PROGRAM VarPersistentes
VAR
		Datos_persistentes :WritePersistentData;
		StartON:TON;
		IntervalON:TON;
END_VAR
VAR // added by the converter: edge detectors and wires of the graphical bodies
    _rt1 : R_TRIG;
END_VAR

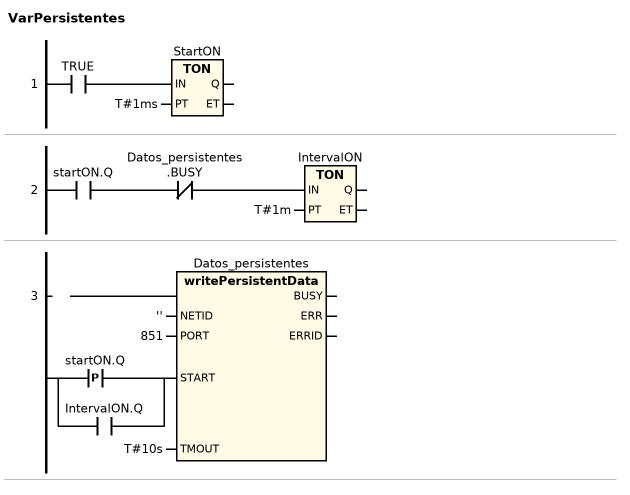
// NETWORK 1
StartON(IN := TRUE, PT := T#1ms); // TON

// NETWORK 2
IntervalON(IN := startON.Q AND NOT Datos_persistentes.BUSY, PT := T#1m); // TON

// NETWORK 3
_rt1(CLK := startON.Q);
Datos_persistentes(NETID := '', PORT := 851, START := _rt1.Q OR IntervalON.Q, TMOUT := T#10s); // writePersistentData

END_PROGRAM

(* stored: Version 1.1.0.1, ProductVersion 3.1.4024.13
   POU VarPersistentes: Id {c7225a0b-a6d3-4468-bd75-bcd48f1979f8}, SpecialFunc None *)
